{attribute 'qualified_only'}
VAR_GLOBAL
	mb_Input_Coils	:	ARRAY [0..3] OF BOOL;
 	mb_Output_Coils	:   ARRAY [0..5] OF BOOL;
	
	iState 			: 	INT;
END_VAR

(* stored: Version 1.1.0.1, ProductVersion 3.1.4024.12
   GVL GVL: Id {c47e991f-c8a6-48c3-a4a7-d83427e5e535} *)
